Yaskawa INFORM job: COFNIJ_DRUT.JBI

/JOB
//NAME COFNIJ_DRUT
//POS
///NPOS 0,0,0,0,0,0
//INST
///DATE 2024/09/12 13:35
///ATTR SC,RW
///GROUP1 RB1,BS1
NOP
'WIREFEED INPUT
DOUT OT#(4096) ON
TIMER T=0.80
DOUT OT#(4096) OFF
END
